FUNCTION_BLOCK L3_CompletedPartHDLR (* Basic Function Block Type *)
  (* Standard: 61499-2 *)
  (* Version 0.0, 2014-11-04, EQUEROL, UJI *)
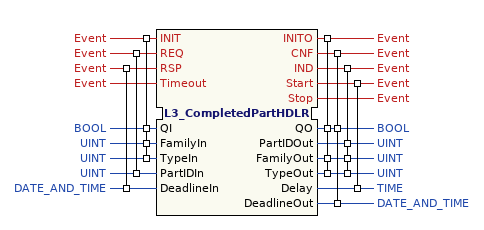
  EVENT_INPUT
    INIT WITH QI, FamilyIn, TypeIn; (* Initialization Request *)
    REQ WITH PartIDIn; (* Normal Execution Request *)
    RSP WITH DeadlineIn; (* Response from OrderManager *)
    Timeout; (* Timeout *)
  END_EVENT
  EVENT_OUTPUT
    INITO WITH QO, FamilyOut, TypeOut; (* Initialization Confirm *)
    CNF WITH QO, DeadlineOut; (* Execution Confirmation *)
    IND WITH PartIDOut, FamilyOut, TypeOut; (* Indication to the OrderManager *)
    Start WITH Delay; (* Timeout start *)
    Stop; (* Timeout stop *)
  END_EVENT
  VAR_INPUT
    QI : BOOL; (* Input event qualifier *)
    FamilyIn : UINT; (* PP Family *)
    TypeIn : UINT; (* PP type *)
    PartIDIn : UINT; (* Completed part identifier *)
    DeadlineIn : DATE_AND_TIME; (* New pp devilery time *)
  END_VAR
  VAR_OUTPUT
    QO : BOOL; (* Output event qualifier *)
    PartIDOut : UINT; (* Part identifier *)
    FamilyOut : UINT; (* PP family *)
    TypeOut : UINT; (* PP type *)
    Delay : TIME; (* Timeout delay *)
    DeadlineOut : DATE_AND_TIME; (* New PP deliverty time *)
  END_VAR
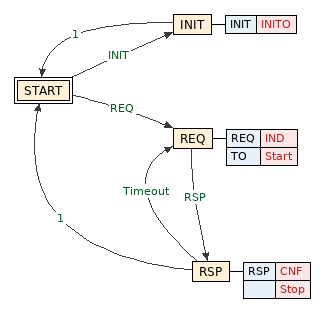
  EC_STATES
    START; (* Initial State *)
    INIT : INIT -> INITO; (* Initialization *)
    REQ : REQ -> IND, TO -> Start; (* Normal execution *)
    RSP : RSP -> CNF, -> Stop;
  END_STATES
  EC_TRANSITIONS
    START TO INIT := INIT;
    INIT TO START := 1;
    START TO REQ := REQ;
    REQ TO RSP := RSP;
    RSP TO START := 1;
    RSP TO REQ := Timeout;
  END_TRANSITIONS
  ALGORITHM INIT IN ST: (* Initialization algorithm *)
IF QI = TRUE THEN
	FamilyOut := FamilyIn;
	TypeOut := TypeIn;
	QO := TRUE;
ELSE
	QO := FALSE;
END_IF;
  END_ALGORITHM
  ALGORITHM REQ IN ST: (* Normally executed algorithm *)
PartIDOut := PartIDIn;
FamilyOut := FamilyIn;
TypeOut := TypeIn;
  END_ALGORITHM
  ALGORITHM RSP IN ST: (* new algorithm *)
DeadlineOut := DeadlineIn;
  END_ALGORITHM
  ALGORITHM TO IN ST: (* TimeOut algo *)
Delay := TIME#1000ms;
  END_ALGORITHM
END_FUNCTION_BLOCK
